FUNCTION_BLOCK FB_Blink
VAR_INPUT
	Mode:INT; //OFF,ON,BLINK
	Duration:TIME;
END_VAR
VAR_OUTPUT
	LED:BOOL;
END_VAR
VAR
	Enable:BOOL;
	Blink_On:BOOL;
	Blink_Off:BOOL;
	SigDown: F_Trig;
	BlinkOn: BOOL;
	BlinkOff: BOOL;
	Down_Timer: TP;
	Up_Timer: TP;
	SigUp: F_Trig;
	
END_VAR
VAR // added by the converter: edge detectors and wires of the graphical bodies
    _w1 : BOOL;
END_VAR

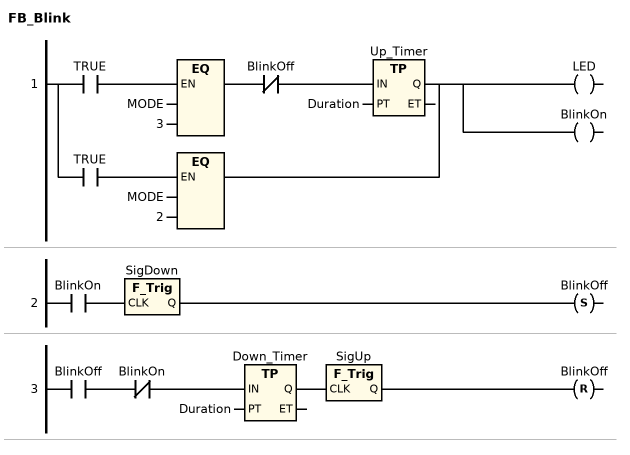
// NETWORK 1
Up_Timer(IN := MODE = 3 AND NOT BlinkOff, PT := Duration); // TP
_w1 := Up_Timer.Q OR MODE = 2;
LED := _w1;
BlinkOn := _w1;

// NETWORK 2
SigDown(CLK := BlinkOn); // F_Trig
BlinkOff S= SigDown.Q;

// NETWORK 3
Down_Timer(IN := BlinkOff AND NOT BlinkOn, PT := Duration); // TP
SigUp(CLK := Down_Timer.Q); // F_Trig
BlinkOff R= SigUp.Q;

END_FUNCTION_BLOCK

(* stored: Version 1.1.0.1, ProductVersion 3.1.4022.18
   POU FB_Blink: Id {9424fac4-64a6-4446-8171-1f45c8338f90}, SpecialFunc None *)
